KUKA KRL data list: chk_w6_ab_ok.dat

&ACCESS RVP2
&COMMENT Condicoes iniciais dock 6 - Deposito
DEFDAT CHK_W6_AB_OK PUBLIC
ENDDAT
